FUNCTION_BLOCK EventOutWrapper_Console (* Composite Function Block Type *)
  (* Standard: 61499-2 *)
  (* Version 0.0, 4/9/2019, erik, nxtControl GmbH, template *)
  PACKAGE Main;
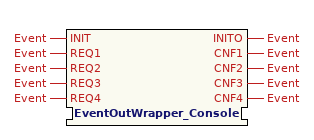
  EVENT_INPUT
    INIT; (* Initialization Request *)
    REQ1; (* Normal Execution Request *)
    REQ2;
    REQ3;
    REQ4;
  END_EVENT
  EVENT_OUTPUT
    INITO; (* Initialization Confirm *)
    CNF1; (* Execution Confirmation *)
    CNF2;
    CNF3;
    CNF4;
  END_EVENT
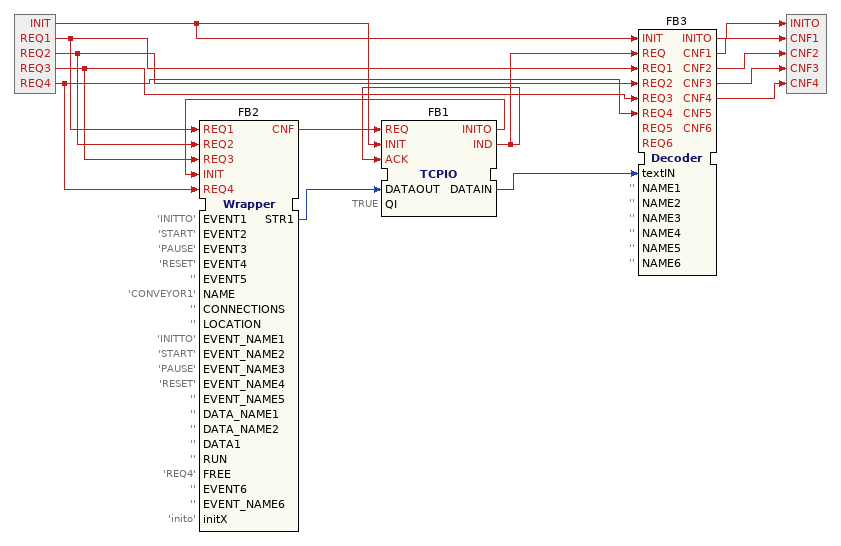
  FBS
    FB1 : TCPIO(QI := TRUE);
    FB2 : Wrapper(EVENT1 := 'INITTO', EVENT2 := 'START', EVENT3 := 'PAUSE', EVENT4 := 'RESET', EVENT5 := '', NAME := 'CONVEYOR1', CONNECTIONS := '', LOCATION := '', EVENT_NAME1 := 'INITTO', EVENT_NAME2 := 'START', EVENT_NAME3 := 'PAUSE', EVENT_NAME4 := 'RESET', EVENT_NAME5 := '', DATA_NAME1 := '', DATA_NAME2 := '', DATA1 := '', RUN := '', FREE := 'REQ4', EVENT6 := '', EVENT_NAME6 := '', initX := 'inito');
    FB3 : Decoder(NAME1 := '', NAME2 := '', NAME3 := '', NAME4 := '', NAME5 := '', NAME6 := '');
  END_FBS
  EVENT_CONNECTIONS
    REQ1 TO FB2.REQ1;
    REQ2 TO FB2.REQ2;
    REQ3 TO FB2.REQ3;
    FB2.CNF TO FB1.REQ;
    INIT TO FB1.INIT;
    FB1.INITO TO FB2.INIT;
    FB1.IND TO FB1.ACK;
    FB1.IND TO FB3.REQ;
    FB3.CNF1 TO CNF1;
    FB3.CNF2 TO CNF2;
    FB3.CNF3 TO CNF3;
    REQ1 TO FB3.REQ1;
    REQ2 TO FB3.REQ2;
    REQ3 TO FB3.REQ3;
    REQ4 TO FB2.REQ4;
    REQ4 TO FB3.REQ4;
    FB3.CNF4 TO CNF4;
    FB3.INITO TO INITO;
    INIT TO FB3.INIT;
  END_CONNECTIONS
  DATA_CONNECTIONS
    FB2.STR1 TO FB1.DATAOUT;
    FB1.DATAIN TO FB3.textIN;
  END_CONNECTIONS
END_FUNCTION_BLOCK
